PROGRAM MAIN
VAR
	StartPb					:	BOOL;
	StopPB					:	BOOL;
	MotorStart				: 	RS;
	Motor					: 	BOOL;
	ProductCnt				: 	CTU;
	LightBarrierSensor		: 	BOOL;
	ProductCounter			: 	WORD;
	TrayChange				: 	BOOL;
END_VAR
VAR // added by the converter: edge detectors and wires of the graphical bodies
    _w1 : ANY;
END_VAR

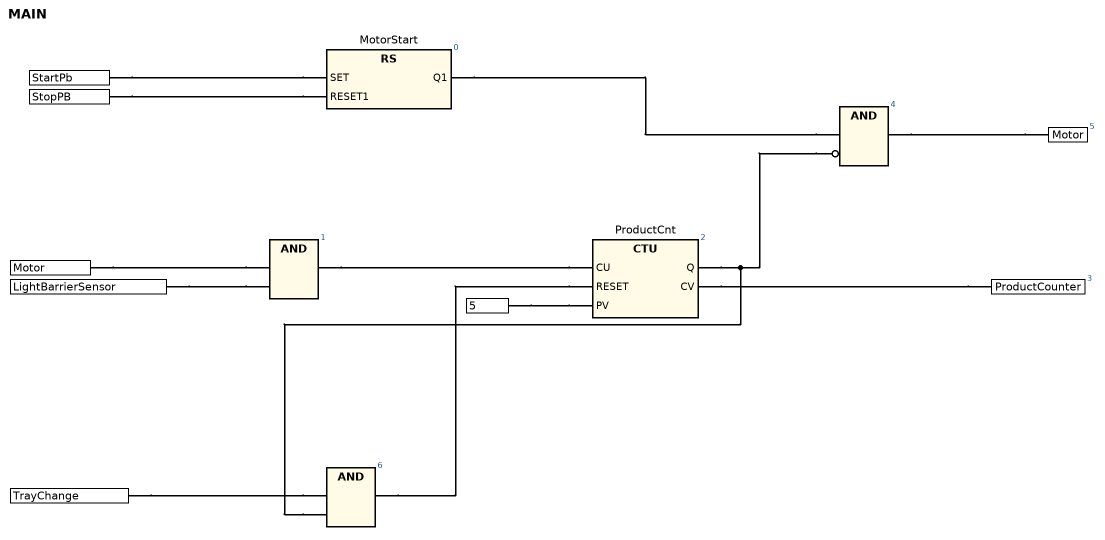
MotorStart(SET := StartPb, RESET1 := StopPB); // RS
ProductCnt(CU := Motor AND LightBarrierSensor, RESET := _w1, PV := 5); // CTU
ProductCounter := ProductCnt.CV;
Motor := MotorStart.Q1 AND NOT ProductCnt.Q;
_w1 := TrayChange AND ProductCnt.Q;

END_PROGRAM

(* stored: Version 1.1.0.1, ProductVersion 3.1.4024.15
   POU MAIN: Id {ccf18a0e-7f61-4b2d-9b0f-37bec9188b76}, SpecialFunc None *)
